# B&R Automation Studio project CITest
Automation Studio 4.5.3.86 SP; technology packages: Acp10Arnc0 5.4.1, mappView 5.4.2

## Configuration ARsim

### Task classes (Cpu.sw)
```
Cyclic#1 (cycle 2000 us, tolerance 0 us):
  main <- Programs.main.prg
  rrbotctrl <- Programs.rrbotctrl.prg
DataObjects: Acp10sys
NcDataObjects: acp10etxen <- MotionObjects.acp10etxen.dob, gConveyora <- MotionObjects.Conveyor.gConveyora.dob, gConveyori <- MotionObjects.Conveyor.gConveyori.dob, gRRBotJ1a <- MotionObjects.RRBotJ1.gRRBotJ1a.dob, gRRBotJ1i <- MotionObjects.RRBotJ1.gRRBotJ1i.dob, gRRBotJ2a <- MotionObjects.RRBotJ2.gRRBotJ2a.dob, gRRBotJ2i <- MotionObjects.RRBotJ2.gRRBotJ2i.dob
Binaries: udbdef, TCData, TCLang, arsvcreg, mvLoader, RRBot, ashwd, User, asfw, arconfig, sysconf, Role, ashwac, iomap, Conveyor, TC, OpcUaMap, acp10cfg, Acp10map
Libraries: operator, runtime, astime, AsIecCon, AsTCP, AsBrStr, AsICMP, Acp10man, Acp10par, NcGlobal, Acp10sim, Acp10_MC, brsystem, sys_lib, MpAxis, MpCom, MpBase, standard, fileio, powerlnk, dataobj
```

### Hardware
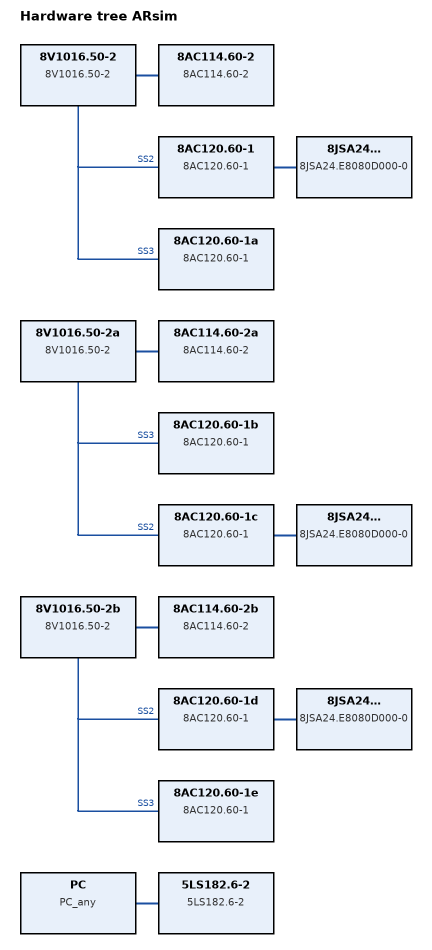
```
5LS182.6-2 : 5LS182.6-2 v1.3.1.0  [SL -> PC.SL1]
8AC114.60-2 : 8AC114.60-2 v1.0.0.8  [SS -> 8V1016.50-2.SS1; PLK1 -> 5LS182.6-2.IF1 [Cable Type=PowerlinkCable, Length=10, Version=1.0.0.2]; PLK2 -> 8AC114.60-2a.PLK1 [Cable Type=PowerlinkCable, Length=10, Version=1.0.0.2]]
8AC114.60-2a : 8AC114.60-2 v1.0.0.8  [SS -> 8V1016.50-2a.SS1; PLK1 -> 8AC114.60-2.PLK2 [Cable Type=PowerlinkCable, Length=10, Version=1.0.0.2]; PLK2 -> 8AC114.60-2b.PLK1 [Cable Type=PowerlinkCable, Length=10, Version=1.0.0.2]]
8AC114.60-2b : 8AC114.60-2 v1.0.0.8  [SS -> 8V1016.50-2b.SS1; PLK1 -> 8AC114.60-2a.PLK2 [Cable Type=PowerlinkCable, Length=10, Version=1.0.0.2]]
8AC120.60-1 : 8AC120.60-1 v2.2.0.0  [SS -> 8V1016.50-2.SS2]
8AC120.60-1a : 8AC120.60-1 v2.2.0.0  [SS -> 8V1016.50-2.SS3]
8AC120.60-1b : 8AC120.60-1 v2.2.0.0  [SS -> 8V1016.50-2a.SS3]
8AC120.60-1c : 8AC120.60-1 v2.2.0.0  [SS -> 8V1016.50-2a.SS2]
8AC120.60-1d : 8AC120.60-1 v2.2.0.0  [SS -> 8V1016.50-2b.SS2]
8AC120.60-1e : 8AC120.60-1 v2.2.0.0  [SS -> 8V1016.50-2b.SS3]
8JSA24.E8080D000-0 : 8JSA24.E8080D000-0 v1.0.6.30  [EC -> 8AC120.60-1.EC; MT -> 8V1016.50-2.MT1]
8JSA24.E8080D000-0a : 8JSA24.E8080D000-0 v1.0.6.30  [EC -> 8AC120.60-1c.EC; MT -> 8V1016.50-2a.MT1]
8JSA24.E8080D000-0b : 8JSA24.E8080D000-0 v1.0.6.30  [EC -> 8AC120.60-1d.EC; MT -> 8V1016.50-2b.MT1]
8V1016.50-2 : 8V1016.50-2 v2.2.0.0
  MotionTP = Acp10Arnc0
  Simulate = standard
  ActiveMotorSimulation_r1 = on
  BothEndSwitchesAreNormallyOpen_r1 = on
  QuickStopIsNormallyOpen_r1 = on
8V1016.50-2a : 8V1016.50-2 v2.2.0.0
  MotionTP = Acp10Arnc0
  Simulate = standard
  ActiveMotorSimulation_r1 = on
  BothEndSwitchesAreNormallyOpen_r1 = on
  QuickStopIsNormallyOpen_r1 = on
8V1016.50-2b : 8V1016.50-2 v2.2.0.0
  MotionTP = Acp10Arnc0
  Simulate = standard
  ActiveMotorSimulation_r1 = on
  BothEndSwitchesAreNormallyOpen_r1 = on
  QuickStopIsNormallyOpen_r1 = on
PC : PC_any v1.1.0.0 (OrderNumber=PC)
  ConfigurationID = ci-test
  SystemTick = 2000
  TaskClassIdleTime = 10000
  Cyclic1Duration = 2000
  Cyclic1Tolerance = 0
  Cyclic1Stack = 65535
  Cyclic2Duration = 20000
  Cyclic2Tolerance = 20000
  Cyclic8Duration = 2000
  Cyclic8Tolerance = 0
  Cyclic8Stack = 65535
  ActivateOpcUa = 1
  OpcUaInformationModels_PV_Version = 1
```

## Logical view

Binary libraries used (declarations not repeated): operator, runtime, astime, AsIecCon, AsTCP, AsBrStr, AsICMP, brsystem, sys_lib, MpCom, standard, MpAxis, MpBase, NcGlobal, Acp10_MC, Acp10man, Acp10par, Acp10sim

### Global.var - Global variables
```iecst
VAR
	joint2PositionDegrees : REAL;
	joint1PositionDegrees : REAL;
	joint1ActualPosition : REAL;
	joint2ActualPosition : REAL;
	joint2SetPosition : REAL;
	joint1SetPosition : REAL;
	redCaseComplete : BOOL;
	greenCaseComplete : BOOL;
	blueCaseComplete : BOOL;
	speakNow : BOOL;
	textCommand : STRING[1000];
	wakeCommand : BOOL;
	TestVar : USINT;
	command : USINT;
	gConveyor : ACP10AXIS_typ;
	gRRBotJ1 : ACP10AXIS_typ;
	gRRBotJ2 : ACP10AXIS_typ;
END_VAR
```

### Package Logical/Libraries - Global libraries

- Visualisation Logical/mappView (not shown)


- Data object Logical/MotionObjects/Conveyor/gConveyora (Apt) (no source held here)

- Data object Logical/MotionObjects/Conveyor/gConveyori (Ax) (no source held here)

- Data object Logical/MotionObjects/RRBotJ1/gRRBotJ1a (Apt) (no source held here)

- Data object Logical/MotionObjects/RRBotJ1/gRRBotJ1i (Ax) (no source held here)

- Data object Logical/MotionObjects/RRBotJ2/gRRBotJ2a (Apt) (no source held here)

- Data object Logical/MotionObjects/RRBotJ2/gRRBotJ2i (Ax) (no source held here)

### Program Logical/Programs/main (IEC)

#### Variables.var
```iecst
VAR
	NextBoxPosition : REAL;
	AutoStep : AutoSteps_enum;
	StartAutoMode : BOOL;
	NextBoxIndex : USINT;
	TON_ShowBox1 : TON;
	TON_ShowBox2 : TON;
	TON_ShowBox3 : TON;
END_VAR
VAR CONSTANT
	EXIT_POSITION : REAL := 8.5;
END_VAR
VAR
	NotifyBox1 : BOOL;
	NotifyBox2 : BOOL;
	NotifyBox3 : BOOL;
END_VAR
VAR CONSTANT
	NOTIFY_POSITION : REAL := 2;
END_VAR
VAR
	TempString : STRING[80];
	BoxPosition1 : REAL;
	BoxPosition2 : REAL;
	BoxPosition3 : REAL;
	WorklightOn : BOOL;
	ShowBox2 : BOOL;
	ShowBox3 : BOOL;
	BoxOffset2 : LREAL;
	BoxOffset3 : LREAL;
	BoxOffset1 : LREAL;
	ShowBox1 : BOOL;
	MotorPosition : REAL;
END_VAR
VAR CONSTANT
	MOTOR_PERIOD : REAL := 2.513;
END_VAR
VAR
	WorklightTransform : STRING[1000];
	Box1Transform : STRING[1000];
	Box2Transform : STRING[1000];
	Box3Transform : STRING[1000];
	Motor1Transform : STRING[1000];
	Motor2Transform : STRING[1000];
	Motor3Transform : STRING[1000];
	Motor4Transform : STRING[1000];
	TotalTransform : STRING[10000];
	PositionString : STRING[80];
	OldParameters : MpAxisBasicParType;
	ConveyorParameters : MpAxisBasicParType;
	Conveyor : MpAxisBasic;
END_VAR
```

#### Main.st
```iecst
PROGRAM _INIT

	Conveyor.MpLink := ADR(gMpLinkConveyor);
	Conveyor.Axis := ADR(gConveyor);
	Conveyor.Enable := TRUE;
	Conveyor.Parameters := ADR(ConveyorParameters);

	ConveyorParameters.Acceleration := 1;
	ConveyorParameters.Deceleration := 1;
	ConveyorParameters.Jog.Acceleration := ConveyorParameters.Acceleration;
	ConveyorParameters.Jog.Deceleration := ConveyorParameters.Deceleration;
	ConveyorParameters.Jog.Velocity := 1;
	ConveyorParameters.Velocity := 1;

	TON_ShowBox1.PT := T#1.75s;
	TON_ShowBox2.PT := T#1.75s;
	TON_ShowBox3.PT := T#1.75s;

END_PROGRAM

PROGRAM _CYCLIC

	// Scaling from axis units to HMI: 100 pixels = 1 meter.
	// On our SVG, the outer belt has a diameter of 80 pixels. This means that one rev of the belt => 251.3 pixels => 2.513 meters

	// Initializing our axis
	IF (Conveyor.Active) THEN
		Conveyor.Power := TRUE;
		IF (Conveyor.PowerOn) THEN
			Conveyor.Home := TRUE;
		END_IF
		IF (Conveyor.IsHomed) THEN
			Conveyor.Home := FALSE;
		END_IF
	END_IF
	IF (Conveyor.Info.MoveDone) THEN
		Conveyor.MoveAbsolute := FALSE;
		Conveyor.MoveAdditive := FALSE;
	END_IF

	// Hard-coding this because it was necessary for me
	ConveyorParameters.Velocity := 1.0;

	// Detect parameter changes and update on the fly
	IF (((ConveyorParameters.Velocity <> OldParameters.Velocity) OR (ConveyorParameters.Acceleration <> OldParameters.Acceleration) OR
		(ConveyorParameters.Deceleration <> OldParameters.Deceleration)) AND (Conveyor.MoveActive)) THEN
		Conveyor.Update := TRUE;
	END_IF
	IF (Conveyor.UpdateDone) THEN
		Conveyor.Update := FALSE;
	END_IF
	OldParameters := ConveyorParameters;

	CASE AutoStep OF
		STEP_IDLE:
			IF (StartAutoMode) THEN
				ShowBox1 := TRUE;
				NextBoxIndex := 1;
				Conveyor.MoveVelocity := TRUE;
				AutoStep := STEP_AUTO;
			END_IF

		STEP_AUTO:
			IF (NOT StartAutoMode) THEN
				Conveyor.MoveVelocity := FALSE;
				AutoStep := STEP_IDLE;
			ELSIF (NextBoxPosition > 3) THEN
				IF (NextBoxIndex = 1) THEN
					ShowBox2 := TRUE;
				ELSIF (NextBoxIndex = 2) THEN
					ShowBox3 := TRUE;
				ELSIF (NextBoxIndex = 3) THEN
					ShowBox1 := TRUE;
				END_IF
				NextBoxIndex := NextBoxIndex + 1;
			END_IF

	END_CASE

	IF (NextBoxIndex = 1) THEN
		NextBoxPosition := BoxPosition1;
	ELSIF (NextBoxIndex = 2) THEN
		NextBoxPosition := BoxPosition2;
	ELSIF (NextBoxIndex = 3) THEN
		NextBoxPosition := BoxPosition3;
	END_IF

	// Handling the motion of the motors
	IF (Conveyor.IsHomed) THEN
		// Logic to figure out where the motors are
		//	MotorPosition := (360 * fmod(LREAL_TO_REAL(Conveyor.Position),MOTOR_PERIOD) / MOTOR_PERIOD);
		MotorPosition := (360 * LREAL_TO_REAL(Conveyor.Position) / MOTOR_PERIOD);
		brsftoa(MotorPosition,ADR(PositionString));
		Motor1Transform := '{"select":"#motorAxis1","duration":2,"spin":[';
		brsstrcat(ADR(Motor1Transform),ADR(PositionString));
		brsstrcat(ADR(Motor1Transform),ADR(',0,0]}'));
		Motor2Transform := '{"select":"#motorAxis2","duration":2,"spin":[';
		brsstrcat(ADR(Motor2Transform),ADR(PositionString));
		brsstrcat(ADR(Motor2Transform),ADR(',0,0]}'));
		Motor3Transform := '{"select":"#motorAxis3","duration":2,"spin":[';
		brsstrcat(ADR(Motor3Transform),ADR(PositionString));
		brsstrcat(ADR(Motor3Transform),ADR(',0,0]}'));
		Motor4Transform := '{"select":"#motorAxis4","duration":2,"spin":[';
		brsstrcat(ADR(Motor4Transform),ADR(PositionString));
		brsstrcat(ADR(Motor4Transform),ADR(',0,0]}'));
	ELSE
		Motor1Transform := '{"select":"#motorAxis1","duration":2,"spin":[0,0,0]}';
		Motor2Transform := '{"select":"#motorAxis2","duration":2,"spin":[0,0,0]}';
		Motor3Transform := '{"select":"#motorAxis3","duration":2,"spin":[0,0,0]}';
		Motor4Transform := '{"select":"#motorAxis4","duration":2,"spin":[0,0,0]}';
	END_IF

	// Handling the motion of the boxes
	IF (EDGEPOS(ShowBox1)) THEN
		TON_ShowBox1.IN := TRUE;
	END_IF
	IF (TON_ShowBox1.Q) THEN
		TON_ShowBox1.IN := FALSE;
		BoxOffset1 := Conveyor.Position;
	END_IF
	IF (TON_ShowBox1.IN) THEN
		Box1Transform := '{"select":"#box_blue_1","display":true,"duration":1500,"scale":[1.2,1.2],"translate":[0,0]}';
	ELSIF (ShowBox1) THEN
		BoxPosition1 := LREAL_TO_REAL(Conveyor.Position - BoxOffset1);
		Box1Transform := '{"select":"#box_blue_1","display":true,"duration":2,"scale":[1,1],"translate":[';
		brsftoa(LREAL_TO_REAL(BoxPosition1*100),ADR(PositionString));
		brsstrcat(ADR(Box1Transform),ADR(PositionString));
		brsstrcat(ADR(Box1Transform),ADR(',0]}'));
	ELSE
		BoxPosition1 := 0;
		Box1Transform := Box2Transform := '{"select":"#box_blue_1","display":false,"duration":2,"scale":[0.1,0.1],"translate":[40,0]}';
	END_IF
	IF (BoxPosition1 > EXIT_POSITION) THEN
		ShowBox1 := FALSE;
		blueCaseComplete := TRUE;
	END_IF

	IF (EDGEPOS(ShowBox2)) THEN
		TON_ShowBox2.IN := TRUE;
	END_IF
	IF (TON_ShowBox2.Q) THEN
		TON_ShowBox2.IN := FALSE;
		BoxOffset2 := Conveyor.Position;
	END_IF
	IF (TON_ShowBox2.IN) THEN
		Box2Transform := '{"select":"#box_green_2","display":true,"duration":1500,"scale":[1.2,1.2],"translate":[0,0]}';
	ELSIF (ShowBox2) THEN
		BoxPosition2 := LREAL_TO_REAL(Conveyor.Position - BoxOffset2);
		Box2Transform := '{"select":"#box_green_2","display":true,"duration":2,"scale":[1,1],"translate":[';
		brsftoa(LREAL_TO_REAL(BoxPosition2*100),ADR(PositionString));
		brsstrcat(ADR(Box2Transform),ADR(PositionString));
		brsstrcat(ADR(Box2Transform),ADR(',0]}'));
	ELSE
		BoxPosition2 := 0;
		Box2Transform := '{"select":"#box_green_2","display":false,"duration":2,"scale":[0.1,0.1],"translate":[30,0]}';
	END_IF

	IF (BoxPosition2 > EXIT_POSITION) THEN
		ShowBox2 := FALSE;
		greenCaseComplete := TRUE;
	END_IF

	IF (EDGEPOS(ShowBox3)) THEN
		TON_ShowBox3.IN := TRUE;
	END_IF
	IF (TON_ShowBox3.Q) THEN
		TON_ShowBox3.IN := FALSE;
		BoxOffset3 := Conveyor.Position;
	END_IF
	IF (TON_ShowBox3.IN) THEN
		Box3Transform := '{"select":"#box_red_3","display":true,"duration":1500,"scale":[1.2,1.2],"translate":[0,0]}';
	ELSIF (ShowBox3) THEN
		BoxPosition3 := LREAL_TO_REAL(Conveyor.Position - BoxOffset3);
		Box3Transform := '{"select":"#box_red_3","display":true,"duration":2,"scale":[1,1],"translate":[';
		brsftoa(LREAL_TO_REAL(BoxPosition3*100),ADR(PositionString));
		brsstrcat(ADR(Box3Transform),ADR(PositionString));
		brsstrcat(ADR(Box3Transform),ADR(',0]}'));
	ELSE
		BoxPosition3 := 0;
		Box3Transform := '{"select":"#box_red_3","display":false,"duration":2,"scale":[0.1,0.1],"translate":[30,0]}';
	END_IF
	IF (BoxPosition3 > EXIT_POSITION) THEN
		ShowBox3 := FALSE;
		redCaseComplete := TRUE;
	END_IF

	// Handling the light
	IF (WorklightOn) THEN
		WorklightTransform := '{"select":"#work_light_beam","display":true,"duration":2,"translate":[0,0]}';
	ELSE
		WorklightTransform := '{"select":"#work_light_beam","display":false,"duration":2,"translate":[0,0]}';
	END_IF

	// Creating the transform string from all elements
	TotalTransform := '[';
	brsstrcat(ADR(TotalTransform),ADR(WorklightTransform));
	brsstrcat(ADR(TotalTransform),ADR(','));
	brsstrcat(ADR(TotalTransform),ADR(Box1Transform));
	brsstrcat(ADR(TotalTransform),ADR(','));
	brsstrcat(ADR(TotalTransform),ADR(Box2Transform));
	brsstrcat(ADR(TotalTransform),ADR(','));
	brsstrcat(ADR(TotalTransform),ADR(Box3Transform));
	brsstrcat(ADR(TotalTransform),ADR(','));
	brsstrcat(ADR(TotalTransform),ADR(Motor1Transform));
	brsstrcat(ADR(TotalTransform),ADR(','));
	brsstrcat(ADR(TotalTransform),ADR(Motor2Transform));
	brsstrcat(ADR(TotalTransform),ADR(','));
	brsstrcat(ADR(TotalTransform),ADR(Motor3Transform));
	brsstrcat(ADR(TotalTransform),ADR(','));
	brsstrcat(ADR(TotalTransform),ADR(Motor4Transform));
	brsstrcat(ADR(TotalTransform),ADR(']'));

	// Calling the FBs
	Conveyor();
	TON_ShowBox1();
	TON_ShowBox2();
	TON_ShowBox3();

END_PROGRAM

PROGRAM _EXIT
	(* Insert code here *)

END_PROGRAM
```

### Program Logical/Programs/rrbotctrl (IEC)

#### Main.st
```iecst
PROGRAM _INIT

	RRBotJ1.Axis := ADR(gRRBotJ1);
	RRBotJ1.MpLink := ADR(gMpLinkRRBotJ1);
	RRBotJ1.Parameters := ADR(RRBotJ1Parameters);
	RRBotJ1.Enable := TRUE;

END_PROGRAM

PROGRAM _CYCLIC

	IF (RRBotJ1.Active) THEN
		RRBotJ1.Power := TRUE;
	END_IF
	IF (RRBotJ1.PowerOn) AND (NOT RRBotJ1.IsHomed) THEN
		RRBotJ1.Home := TRUE;
	END_IF
	IF (RRBotJ1Parameters.Velocity <> OldParameters.Velocity) THEN
		RRBotJ1.Update := TRUE;
	END_IF
	IF (RRBotJ1.UpdateDone) THEN
		RRBotJ1.Update := FALSE;
	END_IF

	RRBotJ1();

	joint1SetPosition := LREAL_TO_REAL((RRBotJ1.Position) * PI / 180);

	joint1ActualPosition := joint1SetPosition;
	joint2ActualPosition;

	OldParameters := RRBotJ1Parameters;

	// Handling the motion of the motors
	IF (RRBotJ1.IsHomed) THEN
		// Logic to figure out where joint 1 is
		joint1Position := REAL_TO_UINT((joint1ActualPosition * 180 / PI) + 180) MOD 360;
		brsitoa(joint1Position,ADR(PositionString));
		joint1Transform := '{"select":"#joint1Group","spin":[';
		brsstrcat(ADR(joint1Transform),ADR(PositionString));
		brsstrcat(ADR(joint1Transform),ADR(',10,0]}'));
		// Logic to figure out where joint 2 is
		joint2Position := REAL_TO_UINT(joint2ActualPosition * 180 / PI) MOD 360;
		brsitoa(joint2Position,ADR(PositionString));
		joint2Transform := '{"select":"#joint2Group","spin":[';
		brsstrcat(ADR(joint2Transform),ADR(PositionString));
		brsstrcat(ADR(joint2Transform),ADR(',10,202]}'));
	ELSE
		joint1Transform := '{"select":"#joint1Group","spin":[0,10,0]}';
		joint2Transform := '{"select":"#joint2Group","spin":[0,10,202]}';
	END_IF

	// Creating the transform string from all elements
	totalTransform := '[';
	brsstrcat(ADR(totalTransform),ADR(joint1Transform));
	brsstrcat(ADR(totalTransform),ADR(','));
	brsstrcat(ADR(totalTransform),ADR(joint2Transform));
	brsstrcat(ADR(totalTransform),ADR(']'));

END_PROGRAM

PROGRAM _EXIT
	(* Insert code here *)

END_PROGRAM
```

Listed in the project but not available here: Logical/Global.typ, Logical/MotionObjects/acp10etxen
